FUNCTION "IterationAndJumpInstructions_GoTo" : Void
{ S7_Optimized_Access := 'true' }
AUTHOR : Myself
FAMILY : SomeFam

   VAR_INPUT
      myCaseSelectorInputVar : DINT;
   END_VAR

   VAR_TEMP
      myVar1 : DINT;   // Comment for my variable 1
      myVar2 : DINT;   // Comment for my variable 2
      myVar3 : DINT;   // Comment for my variable 3
      myVar4 : DINT;   // Comment for my variable 4
   END_VAR

BEGIN

	LocationsAlwaysVisible: //Jump label
	    #myVar1 := 11;

	IF TRUE THEN
	    GOTO LocationsAlwaysVisible;
	END_IF;

END_FUNCTION